// TIA Portal V19 export
TYPE "Prod_Beam_Data"
// stored: Access Published
   STRUCT
      O_ACT : "Prod_Item_small";
      O_TODO { S7_SetPoint := 'True'} : Array[1..15] of "Prod_Item_small";
      O_ENDING { S7_SetPoint := 'True'} : Array[1..5] of "Prod_Item_small";
      O_OUT { S7_SetPoint := 'True'} : Array[1..5] of "Prod_Item_small";
   END_STRUCT;
END_TYPE
